(* Logix 5000 project; controller DispersionPlc vendor 1 type 14 code 108 rev 34.11; software revision 34.01; part 10 of 22 *)
(* tags used below, declared in another part *)
   ONS : BOOL[32];
   T4301Ons : BOOL[32];
   _JISdebug : DINT;
   _Placeholder : DINT;
   AFB : BOOL;
   AFI : BOOL;
   AirMakeup : TIMER;
   AirMakeup_BEAC : ALIAS FOR Local:1:O.Data[12].11;
   Cool_Setpoint_4301 : DINT;
   DispersionAlarms : BOOL[256];
   Emergency_Cool_4301 : BOOL;
   Emergency_Cool_4301_Reset : BOOL;
   Estop_Inx : ALIAS FOR Local:3:I.Data.3;
   Heat_Setpoint_4301 : DINT;
   HS_S51_2 : AStd_DiscreteInput;
   InxAlarms : BOOL[128];
   K2_Temperature_Alarm_Enable_Bit : BOOL;
   LS_T51_High : ALIAS FOR Local:1:I.Data[27].14;
   LVL_W2_High : ALIAS FOR Local:1:I.Data[1].22;
   LVL_W4_High : ALIAS FOR Local:1:I.Data[1].23;
   MaxHeatTmr4301 : TIMER;
   MIXER_A_4301_RUN : ALIAS FOR Local:1:O.Data[0].0;
   MMI_A_4301_01_RUN_PB : BOOL;
   MMI_A_4301_02_RUN_PB : BOOL;
   MMI_AIR_PURGE_4301_PB : BOOL;
   MMI_COOL_DISH_4301_PB : BOOL;
   MMI_COOL_VALVE_4301_PB : BOOL;
   MMI_Dispersion_Interlock_Bypass : BOOL;
   MMI_P_4301_RUN_PB : BOOL;
   MMI_T4301_AIR_PURGE_REQUEST : BOOL;
   MMI_T51_Level : INT;
   MMI_THINNING_LOADING_VALVE : BOOL;
   MMI_XV_4301_PB : BOOL;
   MMI_Z1H_4301_PB : BOOL;
   MMI_Z2H_4301_PB : BOOL;
   MMI_ZH3_4301_PB : BOOL;
   Ones4301 : DINT;
   OneShots2 : DINT;
   PID_T4301C : PID;
   PID_T4301H : PID;
   PS_AirMakeup : ALIAS FOR Local:1:I.Data[33].3;
   RG_T51 : REAL;
   RG_T51_AI_Holding : REAL;
   RG_T51_AI_Raw : INT;
   RG_T51_AI_Samples : DINT;
   RG_T51_Holding1 : REAL;
   RG_T51_Min_Tank_Value : INT;
   RG_T51_OffSet : REAL;
   RG_T51_REMAINDER : REAL;
   RG_T51_Sf : REAL;
   RM_High_Timer : TIMER;
   RM_Pump_P51_Aux : ALIAS FOR Local:1:I.Data[33].2;
   RM_Pump_P51_Run : ALIAS FOR Local:1:O.Data[13].0;
   RM_Pump_P51_Run_PB : ALIAS FOR Local:1:I.Data[40].0;
   RM_Pump_P51_Run_PB_2 : ALIAS FOR Local:1:I.Data[40].2;
   RM_Pump_P51_Stop_PB : ALIAS FOR Local:1:I.Data[40].1;
   RM_Pump_T51_Run_Lamp : ALIAS FOR Local:1:O.Data[12].2;
   RM_Pump_T51_Run_Lamp2 : ALIAS FOR Local:1:O.Data[0].20;
   RM_Tank_T51_Fill_Closed : ALIAS FOR Local:1:O.Data[12].10;
   RM_Tank_T51_Level_Lamp : ALIAS FOR Local:1:O.Data[12].5;
   RM_To_W2 : ALIAS FOR Local:1:I.Data[1].20;
   RM_To_W4 : ALIAS FOR Local:1:I.Data[1].21;
   SP : REAL;
   SPARE_I_1_4_6 : ALIAS FOR Local:1:I.Data[4].6;
   SPARE_O510 : ALIAS FOR Local:5:O.Data.10;
   SPARE_O600 : ALIAS FOR Local:6:O.Data.0;
   SPARE_O601 : ALIAS FOR Local:6:O.Data.1;
   SPARE_O602 : ALIAS FOR Local:6:O.Data.2;
   SPARE_O603 : ALIAS FOR Local:6:O.Data.3;
   SPARE_O604 : ALIAS FOR Local:6:O.Data.4;
   SPARE_O_13_1 : ALIAS FOR Local:13:O.Ch1Data;
   T4301_AIR_PURGE_REQUEST : BOOL;
   T4301_COOLING_OCCURED : BOOL;
   T4301_Cooling_On : BOOL;
   T4301_COOLING_OPERATION : BOOL;
   T4301_COOLING_TEMP : DINT;
   T4301_COOLING_VALVE_HMI : BOOL;
   T4301_DISCHARGE : BOOL;
   T4301_Heating_On : BOOL;
   T4301_HEATING_OPERATION : BOOL;
   T4301_HMI_Cooling : BOOL;
   T4301_HMI_Heating : BOOL;
   T4301_K : Kettle;
   T4301_Manual_AIR_PURGE_REQUEST : BOOL;
   T4301_Mixer : VFD;
   T4301_PID_Setpoints : PID[5];
   T4301_Pids_On : BOOL;
   T4301_PrePurgeTMR : TIMER;
   T4301_Purge_Complete : BOOL;
   T4301_Request_Cooling : BOOL;
   T4301_Request_Cooling_Tmr : TIMER[5];
   T4301_Request_Heating : BOOL;
   T4301_Request_Heating_Hold : BOOL;
   T4301_Request_Heating_Tmr : TIMER[5];
   T4301_Stop_Pids : BOOL;
   T4301ons2 : DINT;
   T4301Purge : Seq64;
   T51_Tank_Max_Lbs : REAL;
   TE_4301A : ALIAS FOR Local:8:I.Ch0Data;
   TempDifferenceCooling4301 : DINT;
   TempDifferenceCooling4301TMR : TIMER;
   testons : DINT;
   THINONS1 : BOOL;
   TOGGLE : BOOL;
   TRANS_PUMP_P_4301_RUN : ALIAS FOR Local:1:O.Data[0].1;
   W2_High_Level : BOOL;
   W4_High_Level : BOOL;
   XV_4301 : ALIAS FOR Local:5:O.Data.0;
   XV_S51_1 : AStd_VlvOC;
   XV_S51_4 : AStd_VlvOC;
(* MainProgram, continued *)

ROUTINE T4301   (* ladder *)
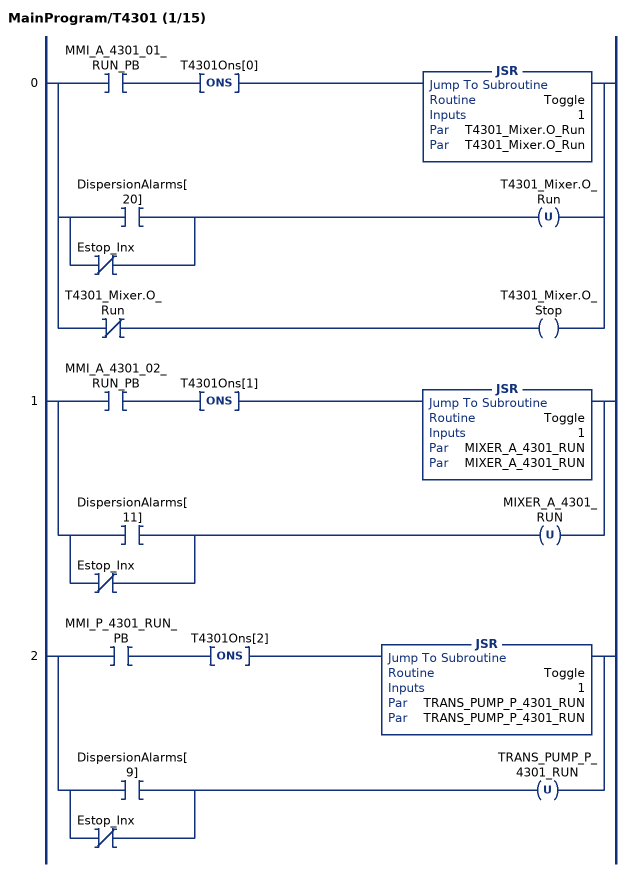
   0: [XIC(MMI_A_4301_01_RUN_PB) ONS(T4301Ons[0]) JSR(Toggle,1,T4301_Mixer.O_Run,T4301_Mixer.O_Run) ,[XIC(DispersionAlarms[20]) ,XIO(Estop_Inx) ] OTU(T4301_Mixer.O_Run) ,XIO(T4301_Mixer.O_Run) OTE(T4301_Mixer.O_Stop) ];
   1: [XIC(MMI_A_4301_02_RUN_PB) ONS(T4301Ons[1]) JSR(Toggle,1,MIXER_A_4301_RUN,MIXER_A_4301_RUN) ,[XIC(DispersionAlarms[11]) ,XIO(Estop_Inx) ] OTU(MIXER_A_4301_RUN) ];
   2: [XIC(MMI_P_4301_RUN_PB) ONS(T4301Ons[2]) JSR(Toggle,1,TRANS_PUMP_P_4301_RUN,TRANS_PUMP_P_4301_RUN) ,[XIC(DispersionAlarms[9]) ,XIO(Estop_Inx) ] OTU(TRANS_PUMP_P_4301_RUN) ];
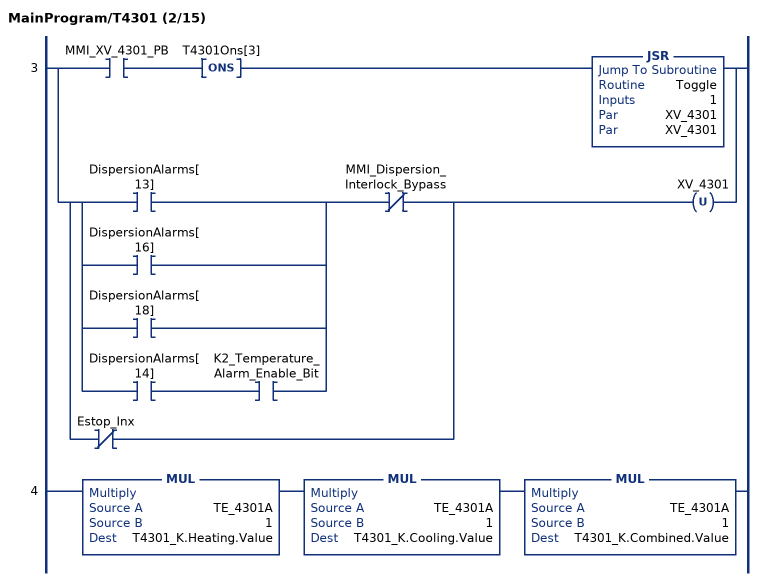
   3: [XIC(MMI_XV_4301_PB) ONS(T4301Ons[3]) JSR(Toggle,1,XV_4301,XV_4301) ,[[XIC(DispersionAlarms[13]) ,XIC(DispersionAlarms[16]) ,XIC(DispersionAlarms[18]) ,XIC(DispersionAlarms[14]) XIC(K2_Temperature_Alarm_Enable_Bit) ] XIO(MMI_Dispersion_Interlock_Bypass) ,XIO(Estop_Inx) ] OTU(XV_4301) ];
   4: MUL(TE_4301A,1,T4301_K.Heating.Value)MUL(TE_4301A,1,T4301_K.Cooling.Value)MUL(TE_4301A,1,T4301_K.Combined.Value);
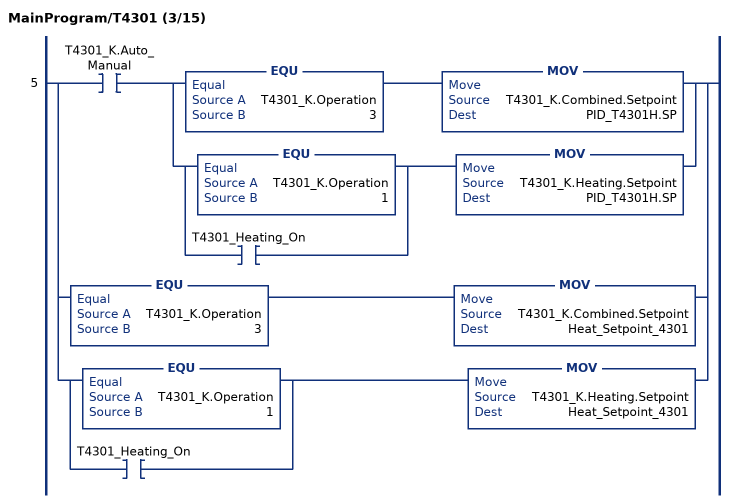
   5: [XIC(T4301_K.Auto_Manual) [EQU(T4301_K.Operation,3) MOV(T4301_K.Combined.Setpoint,PID_T4301H.SP) ,[EQU(T4301_K.Operation,1) ,XIC(T4301_Heating_On) ] MOV(T4301_K.Heating.Setpoint,PID_T4301H.SP) ] ,[EQU(T4301_K.Operation,3) MOV(T4301_K.Combined.Setpoint,Heat_Setpoint_4301) ,[EQU(T4301_K.Operation,1) ,XIC(T4301_Heating_On) ] MOV(T4301_K.Heating.Setpoint,Heat_Setpoint_4301) ] ];
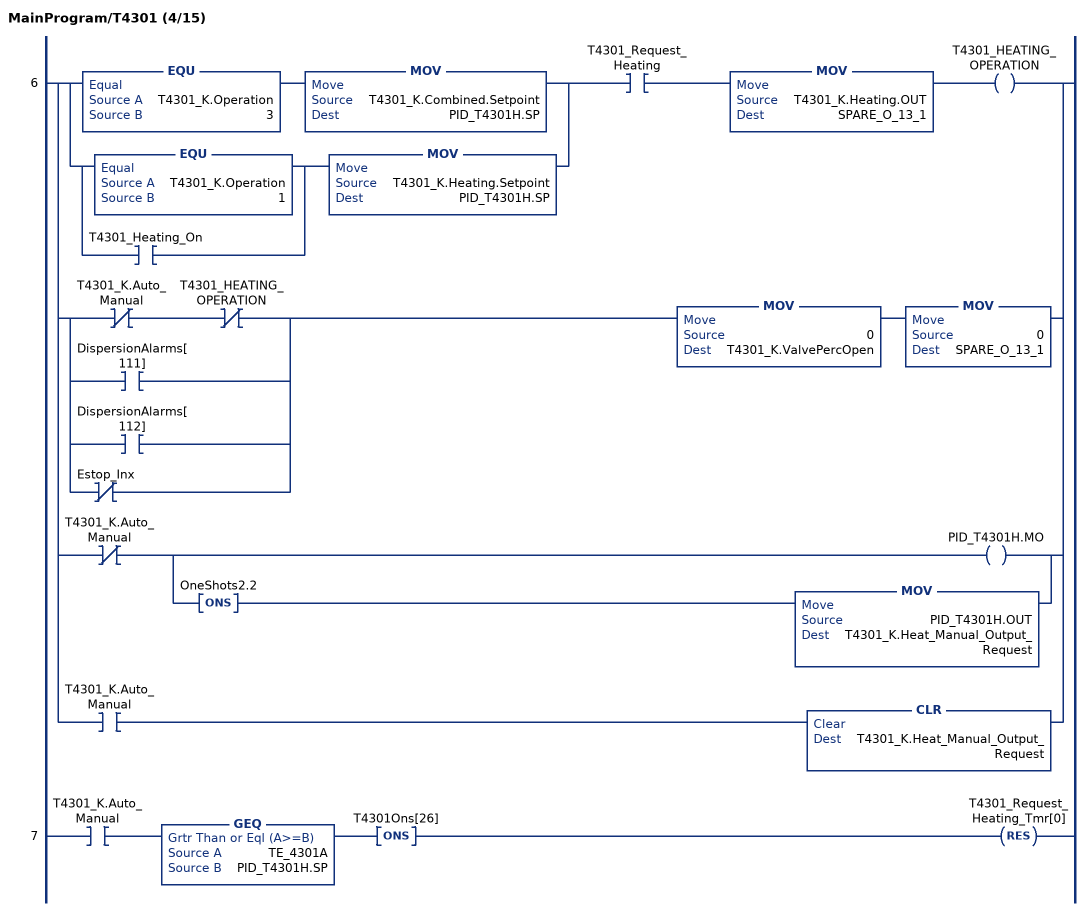
   6: [[EQU(T4301_K.Operation,3) MOV(T4301_K.Combined.Setpoint,PID_T4301H.SP) ,[EQU(T4301_K.Operation,1) ,XIC(T4301_Heating_On) ] MOV(T4301_K.Heating.Setpoint,PID_T4301H.SP) ] XIC(T4301_Request_Heating) MOV(T4301_K.Heating.OUT,SPARE_O_13_1) OTE(T4301_HEATING_OPERATION) ,[XIO(T4301_K.Auto_Manual) XIO(T4301_HEATING_OPERATION) ,[XIC(DispersionAlarms[111]) ,XIC(DispersionAlarms[112]) ,XIO(Estop_Inx) ] ] MOV(0,T4301_K.ValvePercOpen) MOV(0,SPARE_O_13_1) ,[XIO(T4301_K.Auto_Manual) [OTE(PID_T4301H.MO) ,ONS(OneShots2.2) MOV(PID_T4301H.OUT,T4301_K.Heat_Manual_Output_Request) ] ,XIC(T4301_K.Auto_Manual) CLR(T4301_K.Heat_Manual_Output_Request) ] ];
   7: XIC(T4301_K.Auto_Manual)GEQ(TE_4301A,PID_T4301H.SP)ONS(T4301Ons[26])RES(T4301_Request_Heating_Tmr[0]);
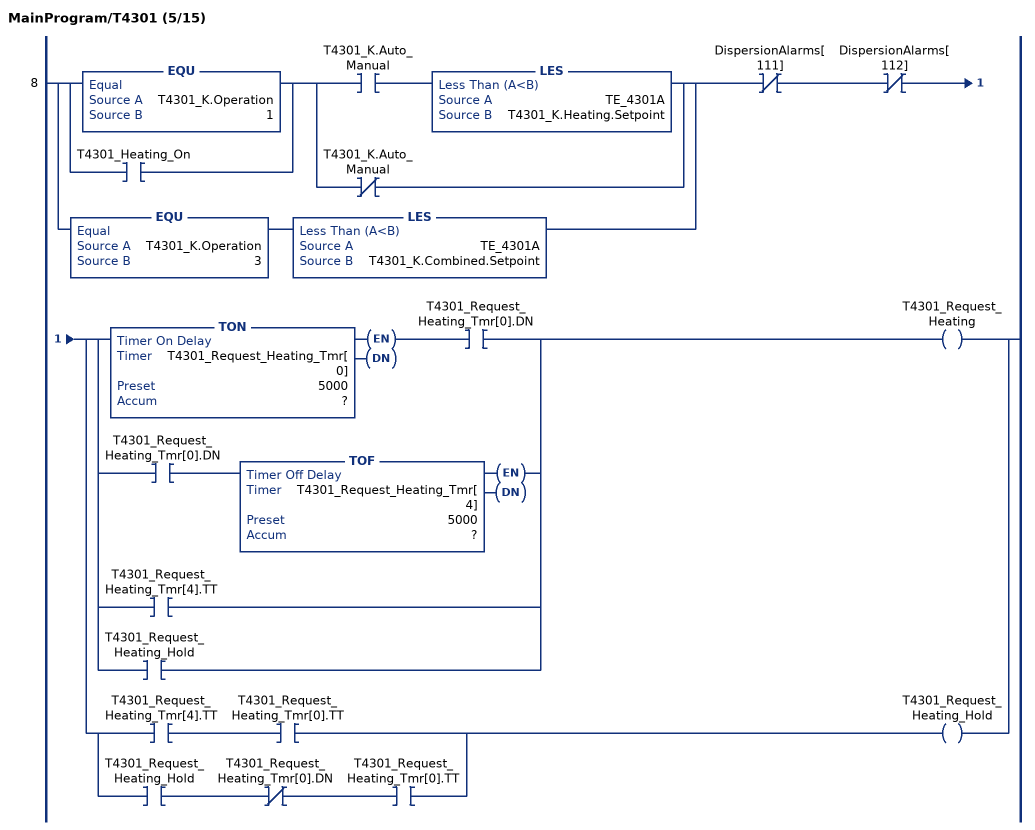
   8: [[EQU(T4301_K.Operation,1) ,XIC(T4301_Heating_On) ] [XIC(T4301_K.Auto_Manual) LES(TE_4301A,T4301_K.Heating.Setpoint) ,XIO(T4301_K.Auto_Manual) ] ,EQU(T4301_K.Operation,3) LES(TE_4301A,T4301_K.Combined.Setpoint) ]XIO(DispersionAlarms[111])XIO(DispersionAlarms[112])[[TON(T4301_Request_Heating_Tmr[0],?,?) XIC(T4301_Request_Heating_Tmr[0].DN) ,XIC(T4301_Request_Heating_Tmr[0].DN) TOF(T4301_Request_Heating_Tmr[4],?,?) ,XIC(T4301_Request_Heating_Tmr[4].TT) ,XIC(T4301_Request_Heating_Hold) ] OTE(T4301_Request_Heating) ,[XIC(T4301_Request_Heating_Tmr[4].TT) XIC(T4301_Request_Heating_Tmr[0].TT) ,XIC(T4301_Request_Heating_Hold) XIO(T4301_Request_Heating_Tmr[0].DN) XIC(T4301_Request_Heating_Tmr[0].TT) ] OTE(T4301_Request_Heating_Hold) ];
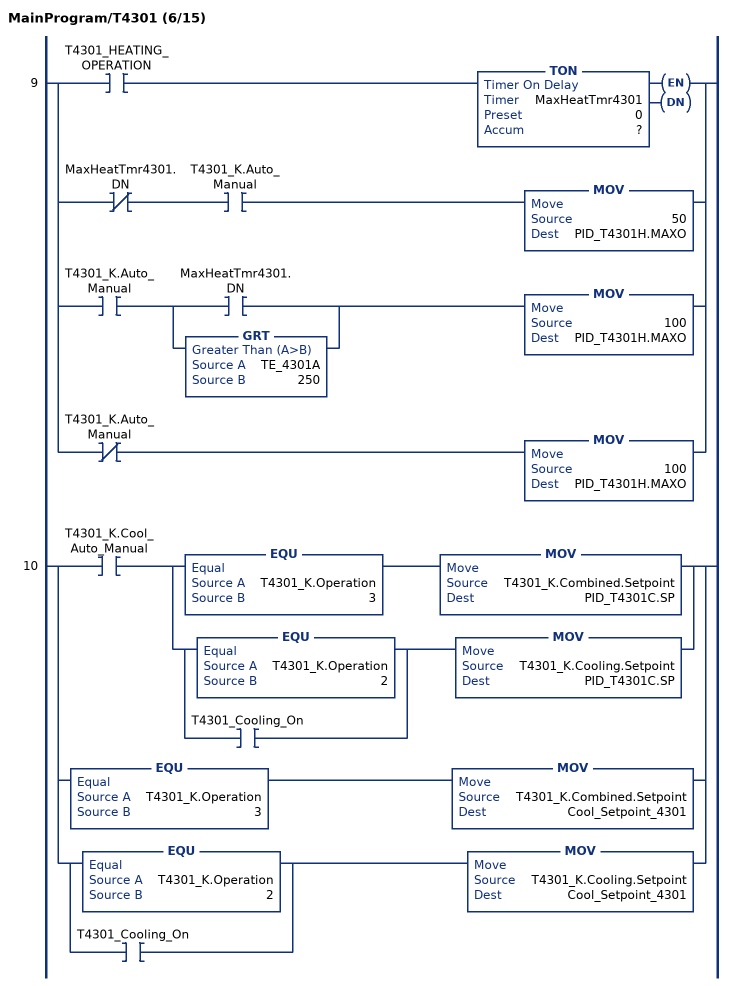
   9: [XIC(T4301_HEATING_OPERATION) TON(MaxHeatTmr4301,?,?) ,XIO(MaxHeatTmr4301.DN) XIC(T4301_K.Auto_Manual) MOV(50,PID_T4301H.MAXO) ,XIC(T4301_K.Auto_Manual) [XIC(MaxHeatTmr4301.DN) ,GRT(TE_4301A,250) ] MOV(100,PID_T4301H.MAXO) ,XIO(T4301_K.Auto_Manual) MOV(100,PID_T4301H.MAXO) ];
   10: [XIC(T4301_K.Cool_Auto_Manual) [EQU(T4301_K.Operation,3) MOV(T4301_K.Combined.Setpoint,PID_T4301C.SP) ,[EQU(T4301_K.Operation,2) ,XIC(T4301_Cooling_On) ] MOV(T4301_K.Cooling.Setpoint,PID_T4301C.SP) ] ,[EQU(T4301_K.Operation,3) MOV(T4301_K.Combined.Setpoint,Cool_Setpoint_4301) ,[EQU(T4301_K.Operation,2) ,XIC(T4301_Cooling_On) ] MOV(T4301_K.Cooling.Setpoint,Cool_Setpoint_4301) ] ];
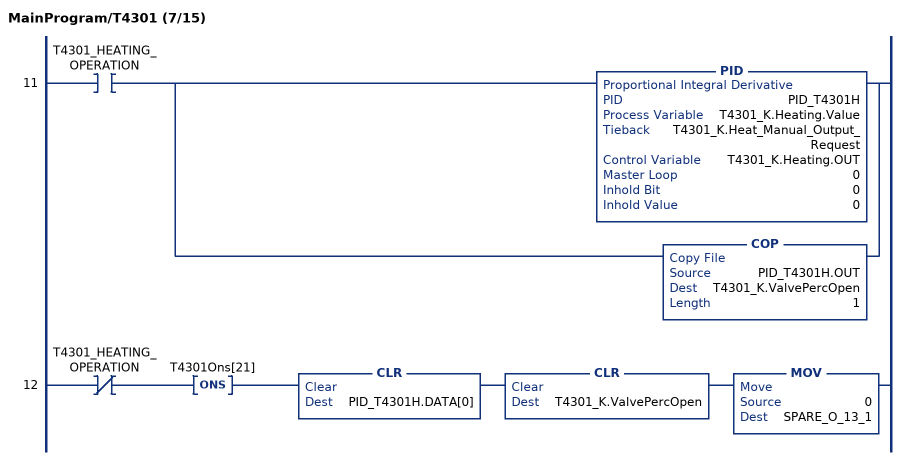
   11: XIC(T4301_HEATING_OPERATION)[PID(PID_T4301H,T4301_K.Heating.Value,T4301_K.Heat_Manual_Output_Request,T4301_K.Heating.OUT,0,0,0) ,COP(PID_T4301H.OUT,T4301_K.ValvePercOpen,1) ];
   12: XIO(T4301_HEATING_OPERATION)ONS(T4301Ons[21])CLR(PID_T4301H.DATA[0])CLR(T4301_K.ValvePercOpen)MOV(0,SPARE_O_13_1);
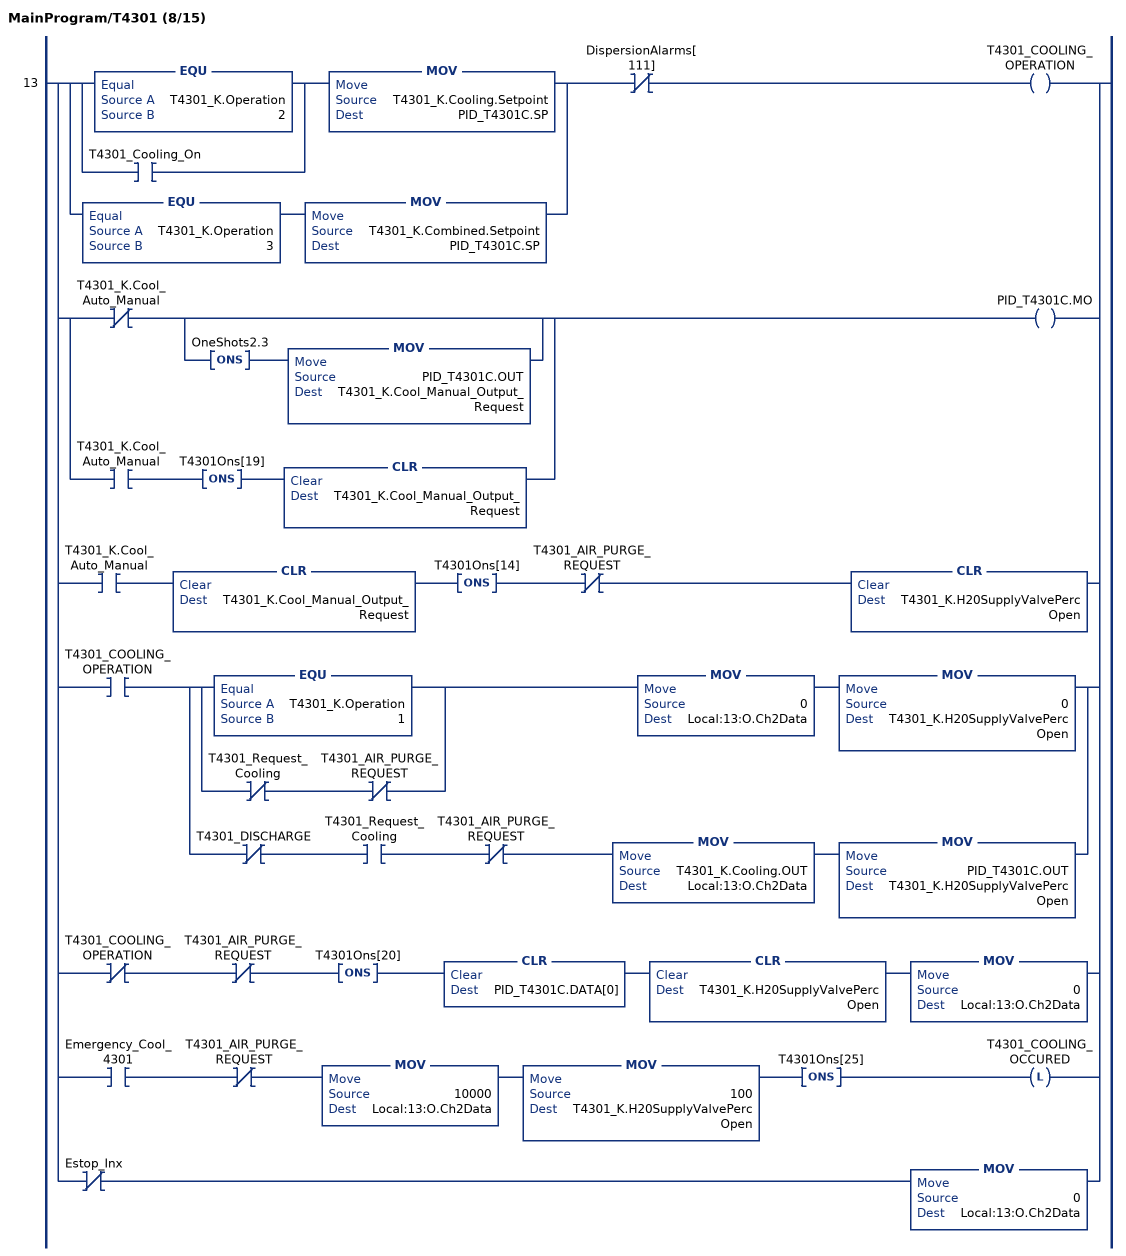
   13: [[[EQU(T4301_K.Operation,2) ,XIC(T4301_Cooling_On) ] MOV(T4301_K.Cooling.Setpoint,PID_T4301C.SP) ,EQU(T4301_K.Operation,3) MOV(T4301_K.Combined.Setpoint,PID_T4301C.SP) ] XIO(DispersionAlarms[111]) OTE(T4301_COOLING_OPERATION) ,[[XIO(T4301_K.Cool_Auto_Manual) [,ONS(OneShots2.3) MOV(PID_T4301C.OUT,T4301_K.Cool_Manual_Output_Request) ] ,XIC(T4301_K.Cool_Auto_Manual) ONS(T4301Ons[19]) CLR(T4301_K.Cool_Manual_Output_Request) ] OTE(PID_T4301C.MO) ,XIC(T4301_K.Cool_Auto_Manual) CLR(T4301_K.Cool_Manual_Output_Request) ONS(T4301Ons[14]) XIO(T4301_AIR_PURGE_REQUEST) CLR(T4301_K.H20SupplyValvePercOpen) ] ,XIC(T4301_COOLING_OPERATION) [[EQU(T4301_K.Operation,1) ,XIO(T4301_Request_Cooling) XIO(T4301_AIR_PURGE_REQUEST) ] MOV(0,Local:13:O.Ch2Data) MOV(0,T4301_K.H20SupplyValvePercOpen) ,XIO(T4301_DISCHARGE) XIC(T4301_Request_Cooling) XIO(T4301_AIR_PURGE_REQUEST) MOV(T4301_K.Cooling.OUT,Local:13:O.Ch2Data) MOV(PID_T4301C.OUT,T4301_K.H20SupplyValvePercOpen) ] ,XIO(T4301_COOLING_OPERATION) XIO(T4301_AIR_PURGE_REQUEST) ONS(T4301Ons[20]) CLR(PID_T4301C.DATA[0]) CLR(T4301_K.H20SupplyValvePercOpen) MOV(0,Local:13:O.Ch2Data) ,XIC(Emergency_Cool_4301) XIO(T4301_AIR_PURGE_REQUEST) MOV(10000,Local:13:O.Ch2Data) MOV(100,T4301_K.H20SupplyValvePercOpen) ONS(T4301Ons[25]) OTL(T4301_COOLING_OCCURED) ,XIO(Estop_Inx) MOV(0,Local:13:O.Ch2Data) ];
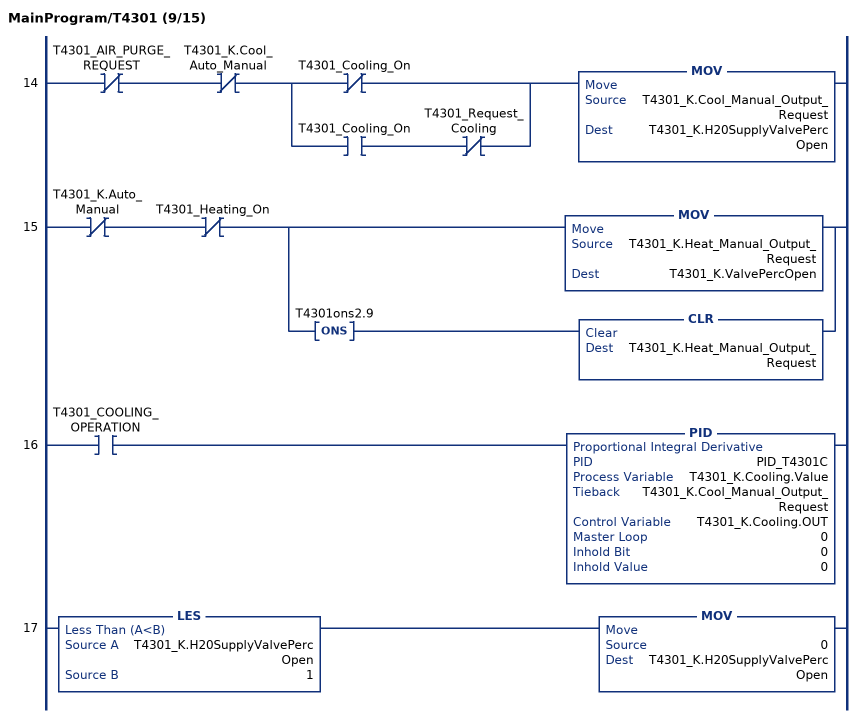
   14: XIO(T4301_AIR_PURGE_REQUEST)XIO(T4301_K.Cool_Auto_Manual)[XIO(T4301_Cooling_On) ,XIC(T4301_Cooling_On) XIO(T4301_Request_Cooling) ]MOV(T4301_K.Cool_Manual_Output_Request,T4301_K.H20SupplyValvePercOpen);
   15: XIO(T4301_K.Auto_Manual)XIO(T4301_Heating_On)[MOV(T4301_K.Heat_Manual_Output_Request,T4301_K.ValvePercOpen) ,ONS(T4301ons2.9) CLR(T4301_K.Heat_Manual_Output_Request) ];
   16: XIC(T4301_COOLING_OPERATION)PID(PID_T4301C,T4301_K.Cooling.Value,T4301_K.Cool_Manual_Output_Request,T4301_K.Cooling.OUT,0,0,0);
   17: LES(T4301_K.H20SupplyValvePercOpen,1)MOV(0,T4301_K.H20SupplyValvePercOpen);
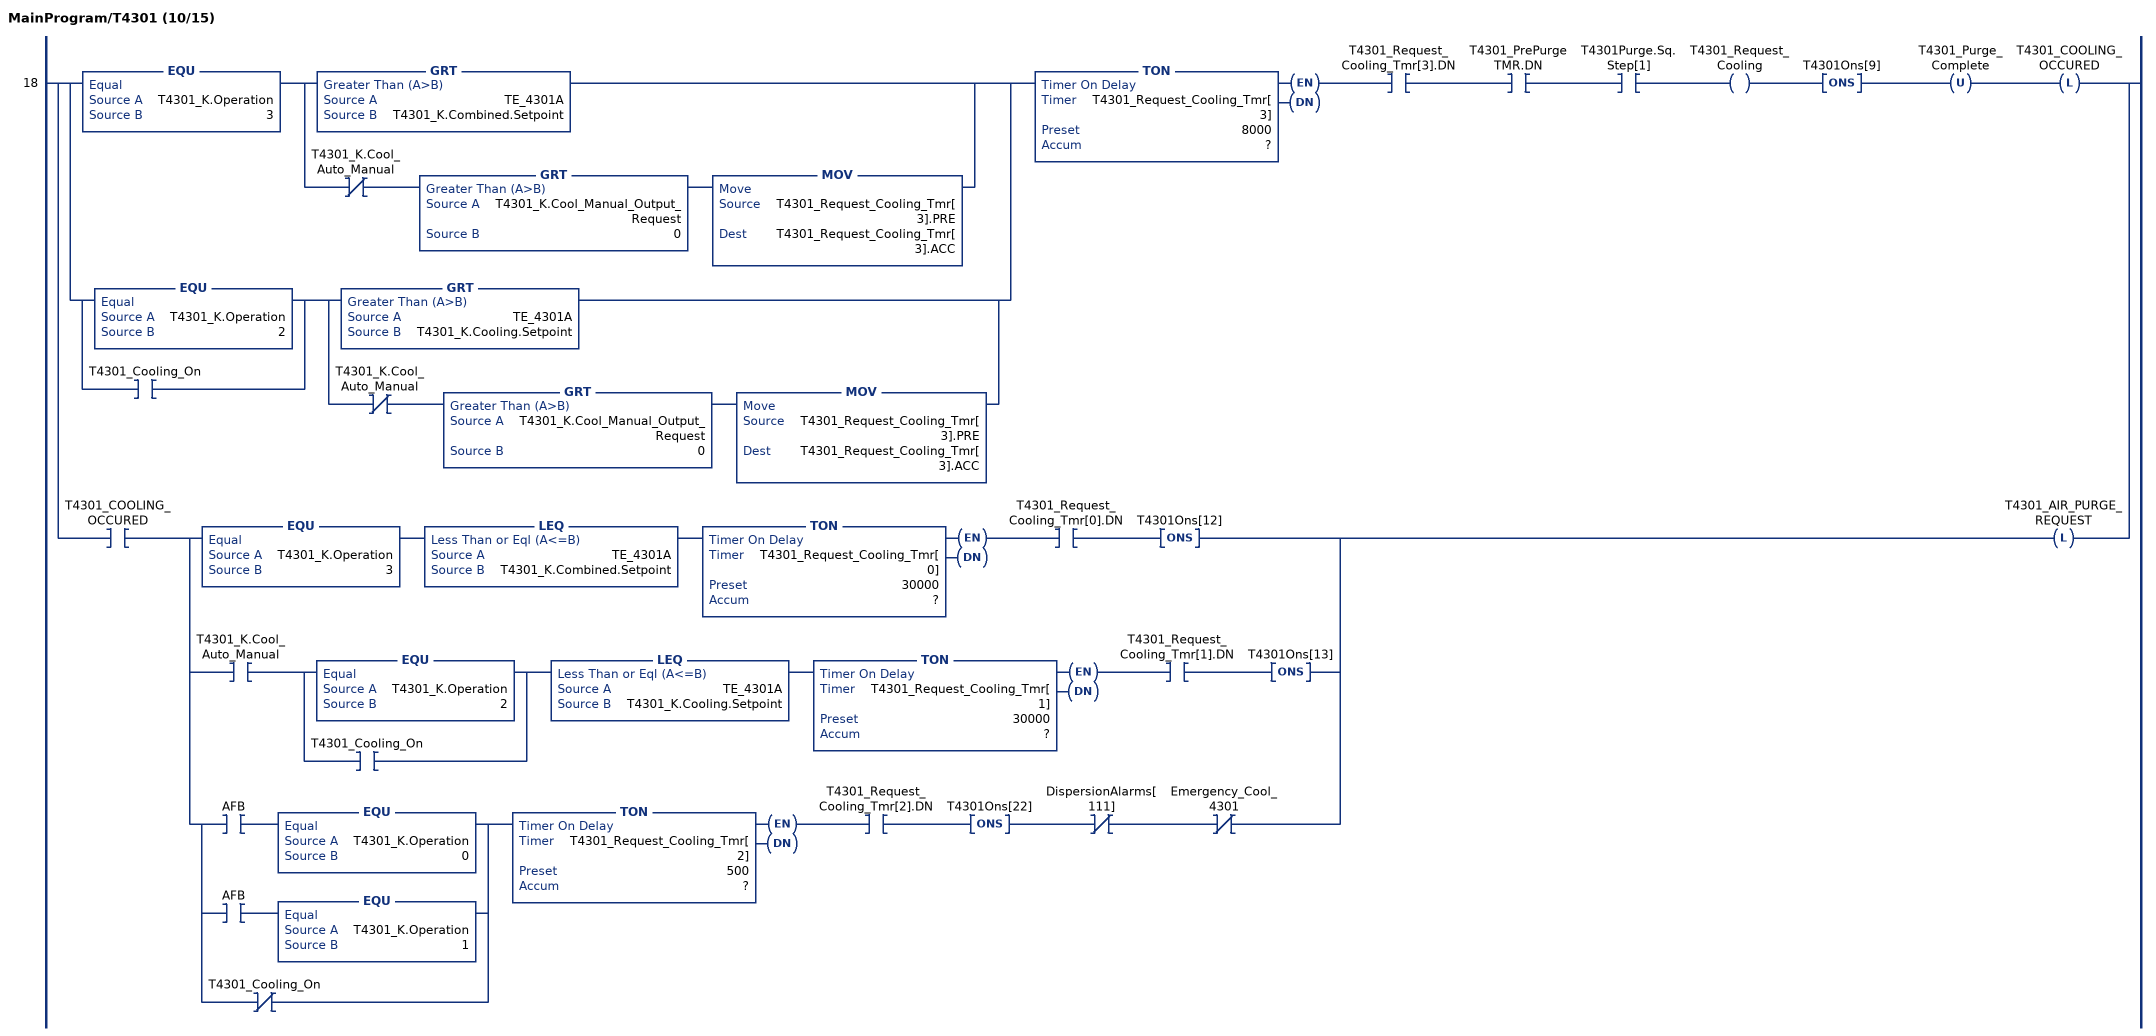
   18: [[EQU(T4301_K.Operation,3) [GRT(TE_4301A,T4301_K.Combined.Setpoint) ,XIO(T4301_K.Cool_Auto_Manual) GRT(T4301_K.Cool_Manual_Output_Request,0) MOV(T4301_Request_Cooling_Tmr[3].PRE,T4301_Request_Cooling_Tmr[3].ACC) ] ,[EQU(T4301_K.Operation,2) ,XIC(T4301_Cooling_On) ] [GRT(TE_4301A,T4301_K.Cooling.Setpoint) ,XIO(T4301_K.Cool_Auto_Manual) GRT(T4301_K.Cool_Manual_Output_Request,0) MOV(T4301_Request_Cooling_Tmr[3].PRE,T4301_Request_Cooling_Tmr[3].ACC) ] ] TON(T4301_Request_Cooling_Tmr[3],?,?) XIC(T4301_Request_Cooling_Tmr[3].DN) XIC(T4301_PrePurgeTMR.DN) XIC(T4301Purge.Sq.Step[1]) OTE(T4301_Request_Cooling) ONS(T4301Ons[9]) OTU(T4301_Purge_Complete) OTL(T4301_COOLING_OCCURED) ,XIC(T4301_COOLING_OCCURED) [EQU(T4301_K.Operation,3) LEQ(TE_4301A,T4301_K.Combined.Setpoint) TON(T4301_Request_Cooling_Tmr[0],?,?) XIC(T4301_Request_Cooling_Tmr[0].DN) ONS(T4301Ons[12]) ,XIC(T4301_K.Cool_Auto_Manual) [EQU(T4301_K.Operation,2) ,XIC(T4301_Cooling_On) ] LEQ(TE_4301A,T4301_K.Cooling.Setpoint) TON(T4301_Request_Cooling_Tmr[1],?,?) XIC(T4301_Request_Cooling_Tmr[1].DN) ONS(T4301Ons[13]) ,[XIC(AFB) EQU(T4301_K.Operation,0) ,XIC(AFB) EQU(T4301_K.Operation,1) ,XIO(T4301_Cooling_On) ] TON(T4301_Request_Cooling_Tmr[2],?,?) XIC(T4301_Request_Cooling_Tmr[2].DN) ONS(T4301Ons[22]) XIO(DispersionAlarms[111]) XIO(Emergency_Cool_4301) ] OTL(T4301_AIR_PURGE_REQUEST) ];
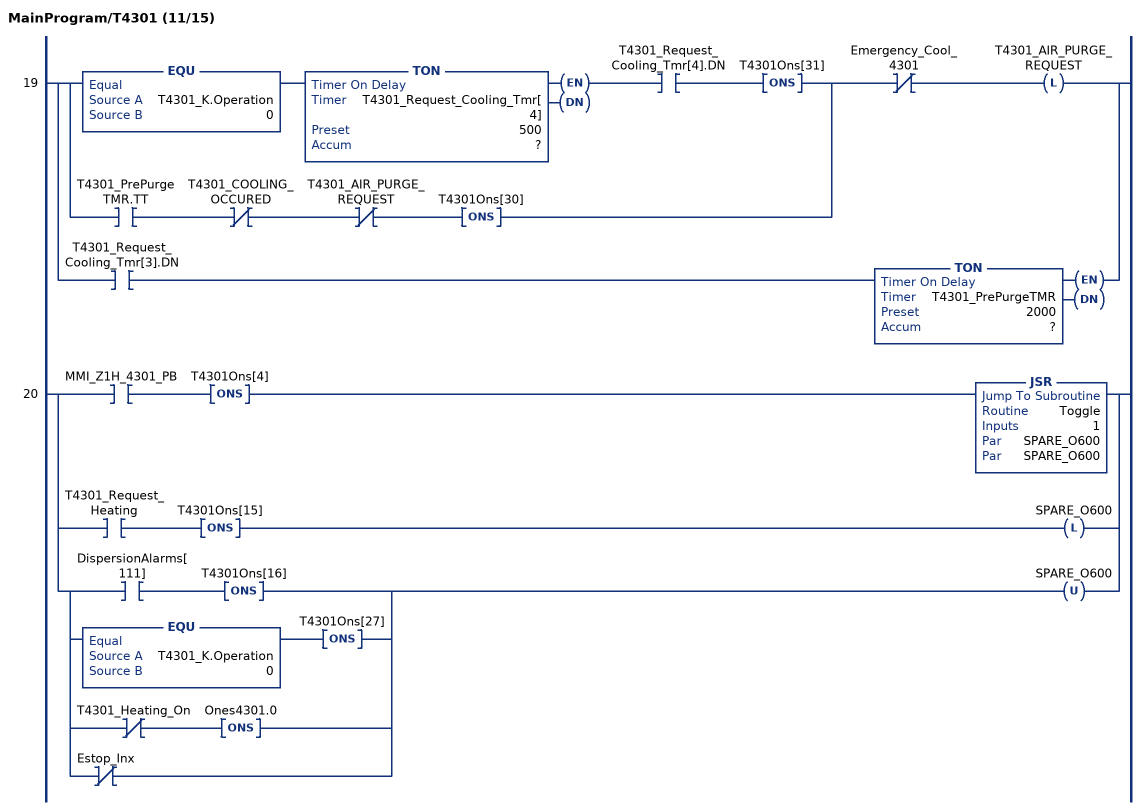
   19: [[EQU(T4301_K.Operation,0) TON(T4301_Request_Cooling_Tmr[4],?,?) XIC(T4301_Request_Cooling_Tmr[4].DN) ONS(T4301Ons[31]) ,XIC(T4301_PrePurgeTMR.TT) XIO(T4301_COOLING_OCCURED) XIO(T4301_AIR_PURGE_REQUEST) ONS(T4301Ons[30]) ] XIO(Emergency_Cool_4301) OTL(T4301_AIR_PURGE_REQUEST) ,XIC(T4301_Request_Cooling_Tmr[3].DN) TON(T4301_PrePurgeTMR,?,?) ];
   20: [XIC(MMI_Z1H_4301_PB) ONS(T4301Ons[4]) JSR(Toggle,1,SPARE_O600,SPARE_O600) ,XIC(T4301_Request_Heating) ONS(T4301Ons[15]) OTL(SPARE_O600) ,[XIC(DispersionAlarms[111]) ONS(T4301Ons[16]) ,[EQU(T4301_K.Operation,0) ONS(T4301Ons[27]) ,XIO(T4301_Heating_On) ONS(Ones4301.0) ] ,XIO(Estop_Inx) ] OTU(SPARE_O600) ];
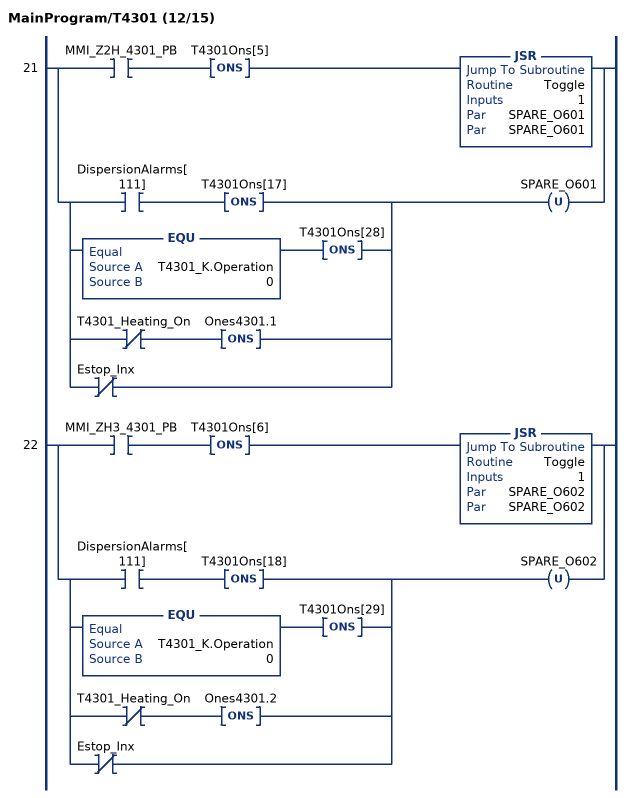
   21: [XIC(MMI_Z2H_4301_PB) ONS(T4301Ons[5]) JSR(Toggle,1,SPARE_O601,SPARE_O601) ,[XIC(DispersionAlarms[111]) ONS(T4301Ons[17]) ,[EQU(T4301_K.Operation,0) ONS(T4301Ons[28]) ,XIO(T4301_Heating_On) ONS(Ones4301.1) ] ,XIO(Estop_Inx) ] OTU(SPARE_O601) ];
   22: [XIC(MMI_ZH3_4301_PB) ONS(T4301Ons[6]) JSR(Toggle,1,SPARE_O602,SPARE_O602) ,[XIC(DispersionAlarms[111]) ONS(T4301Ons[18]) ,[EQU(T4301_K.Operation,0) ONS(T4301Ons[29]) ,XIO(T4301_Heating_On) ONS(Ones4301.2) ] ,XIO(Estop_Inx) ] OTU(SPARE_O602) ];
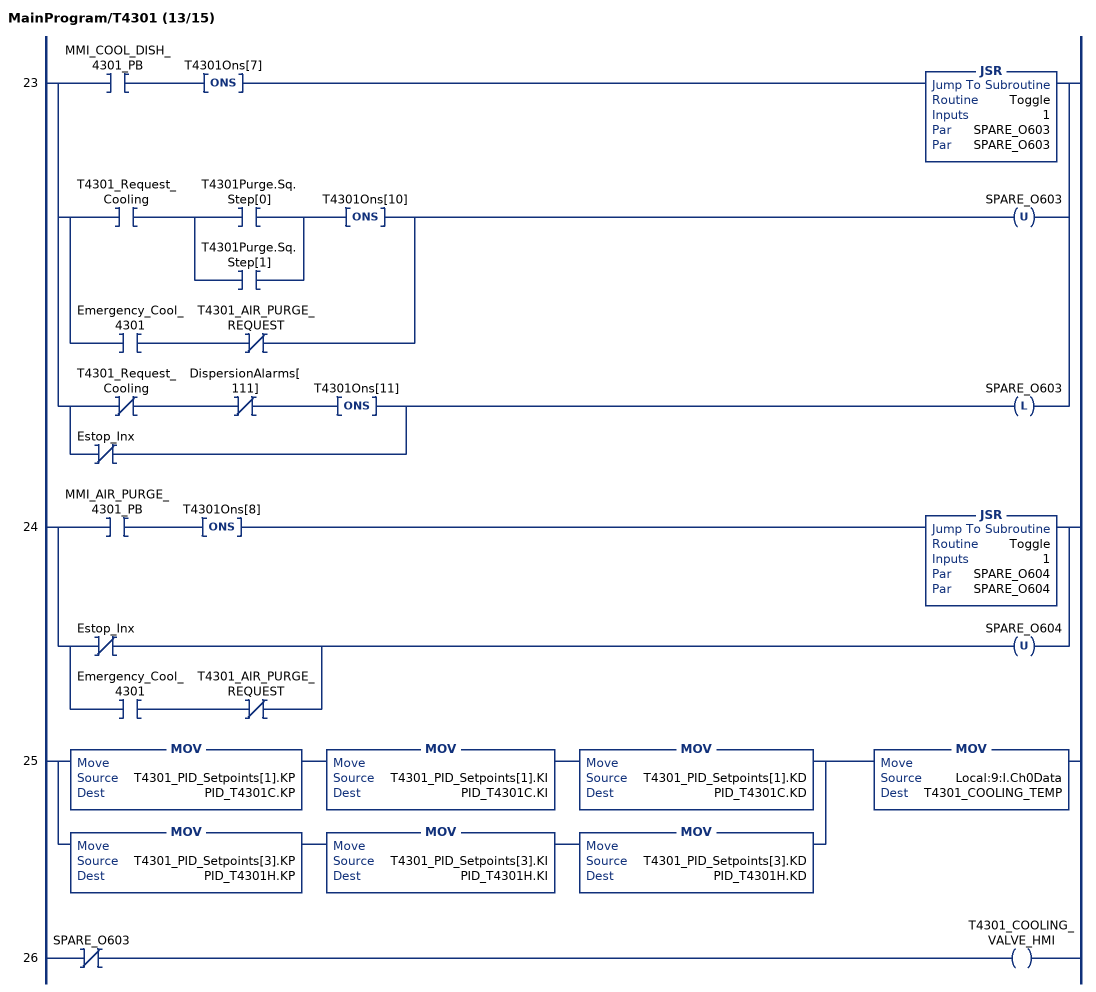
   23: [XIC(MMI_COOL_DISH_4301_PB) ONS(T4301Ons[7]) JSR(Toggle,1,SPARE_O603,SPARE_O603) ,[XIC(T4301_Request_Cooling) [XIC(T4301Purge.Sq.Step[0]) ,XIC(T4301Purge.Sq.Step[1]) ] ONS(T4301Ons[10]) ,XIC(Emergency_Cool_4301) XIO(T4301_AIR_PURGE_REQUEST) ] OTU(SPARE_O603) ,[XIO(T4301_Request_Cooling) XIO(DispersionAlarms[111]) ONS(T4301Ons[11]) ,XIO(Estop_Inx) ] OTL(SPARE_O603) ];
   24: [XIC(MMI_AIR_PURGE_4301_PB) ONS(T4301Ons[8]) JSR(Toggle,1,SPARE_O604,SPARE_O604) ,[XIO(Estop_Inx) ,XIC(Emergency_Cool_4301) XIO(T4301_AIR_PURGE_REQUEST) ] OTU(SPARE_O604) ];
   25: [MOV(T4301_PID_Setpoints[1].KP,PID_T4301C.KP) MOV(T4301_PID_Setpoints[1].KI,PID_T4301C.KI) MOV(T4301_PID_Setpoints[1].KD,PID_T4301C.KD) ,MOV(T4301_PID_Setpoints[3].KP,PID_T4301H.KP) MOV(T4301_PID_Setpoints[3].KI,PID_T4301H.KI) MOV(T4301_PID_Setpoints[3].KD,PID_T4301H.KD) ]MOV(Local:9:I.Ch0Data,T4301_COOLING_TEMP);
   26: XIO(SPARE_O603)OTE(T4301_COOLING_VALVE_HMI);
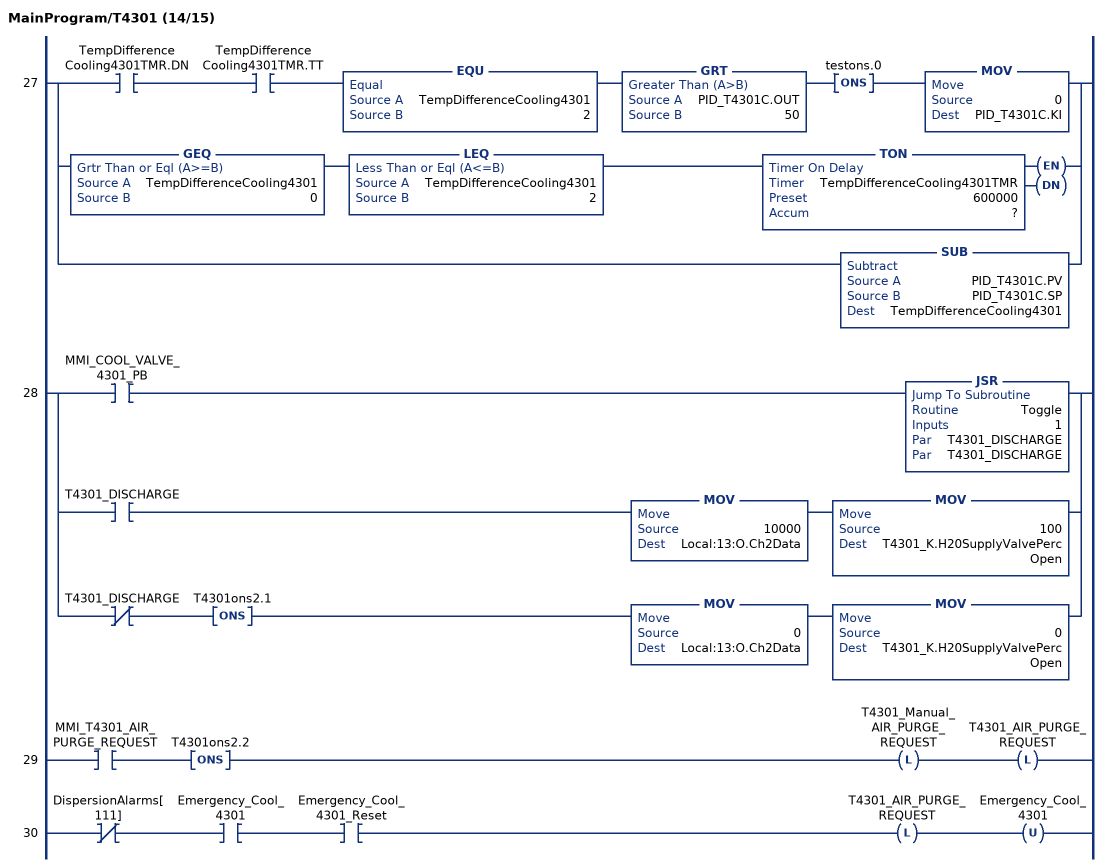
   27: [XIC(TempDifferenceCooling4301TMR.DN) XIC(TempDifferenceCooling4301TMR.TT) EQU(TempDifferenceCooling4301,2) GRT(PID_T4301C.OUT,50) ONS(testons.0) MOV(0,PID_T4301C.KI) ,GEQ(TempDifferenceCooling4301,0) LEQ(TempDifferenceCooling4301,2) TON(TempDifferenceCooling4301TMR,?,?) ,SUB(PID_T4301C.PV,PID_T4301C.SP,TempDifferenceCooling4301) ];
   28: [XIC(MMI_COOL_VALVE_4301_PB) JSR(Toggle,1,T4301_DISCHARGE,T4301_DISCHARGE) ,XIC(T4301_DISCHARGE) MOV(10000,Local:13:O.Ch2Data) MOV(100,T4301_K.H20SupplyValvePercOpen) ,XIO(T4301_DISCHARGE) ONS(T4301ons2.1) MOV(0,Local:13:O.Ch2Data) MOV(0,T4301_K.H20SupplyValvePercOpen) ];
   29: XIC(MMI_T4301_AIR_PURGE_REQUEST)ONS(T4301ons2.2)OTL(T4301_Manual_AIR_PURGE_REQUEST)OTL(T4301_AIR_PURGE_REQUEST);
   30: XIO(DispersionAlarms[111])XIC(Emergency_Cool_4301)XIC(Emergency_Cool_4301_Reset)OTL(T4301_AIR_PURGE_REQUEST)OTU(Emergency_Cool_4301);
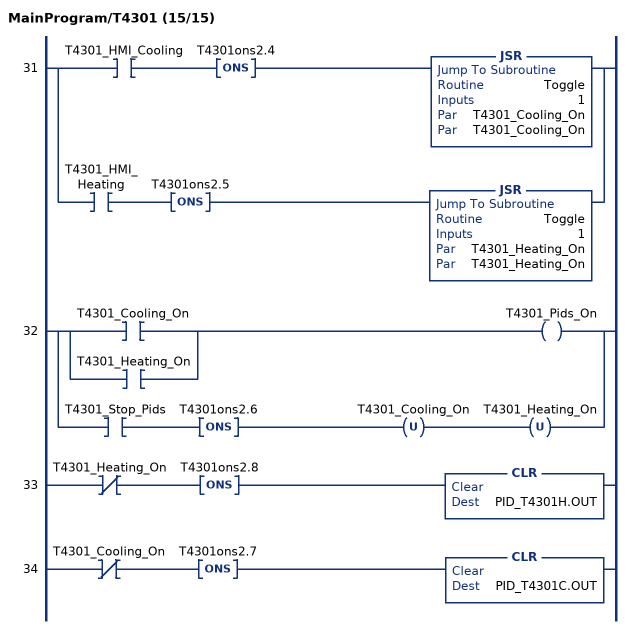
   31: [XIC(T4301_HMI_Cooling) ONS(T4301ons2.4) JSR(Toggle,1,T4301_Cooling_On,T4301_Cooling_On) ,XIC(T4301_HMI_Heating) ONS(T4301ons2.5) JSR(Toggle,1,T4301_Heating_On,T4301_Heating_On) ];
   32: [[XIC(T4301_Cooling_On) ,XIC(T4301_Heating_On) ] OTE(T4301_Pids_On) ,XIC(T4301_Stop_Pids) ONS(T4301ons2.6) OTU(T4301_Cooling_On) OTU(T4301_Heating_On) ];
   33: XIO(T4301_Heating_On)ONS(T4301ons2.8)CLR(PID_T4301H.OUT);
   34: XIO(T4301_Cooling_On)ONS(T4301ons2.7)CLR(PID_T4301C.OUT);
END_ROUTINE

ROUTINE T51   (* ladder *)
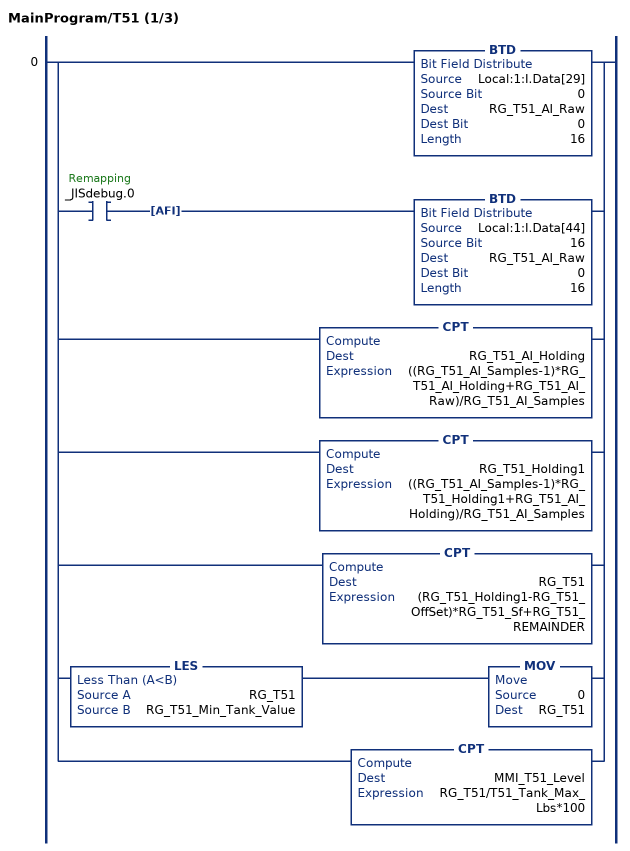
   0: [BTD(Local:1:I.Data[29],0,RG_T51_AI_Raw,0,16) ,XIC(_JISdebug.0) AFI() BTD(Local:1:I.Data[44],16,RG_T51_AI_Raw,0,16) ,CPT(RG_T51_AI_Holding,((RG_T51_AI_Samples-1)*RG_T51_AI_Holding+RG_T51_AI_Raw)/RG_T51_AI_Samples) ,CPT(RG_T51_Holding1,((RG_T51_AI_Samples-1)*RG_T51_Holding1+RG_T51_AI_Holding)/RG_T51_AI_Samples) ,CPT(RG_T51,(RG_T51_Holding1-RG_T51_OffSet)*RG_T51_Sf+RG_T51_REMAINDER) ,LES(RG_T51,RG_T51_Min_Tank_Value) MOV(0,RG_T51) ,CPT(MMI_T51_Level,RG_T51/T51_Tank_Max_Lbs*100) ];
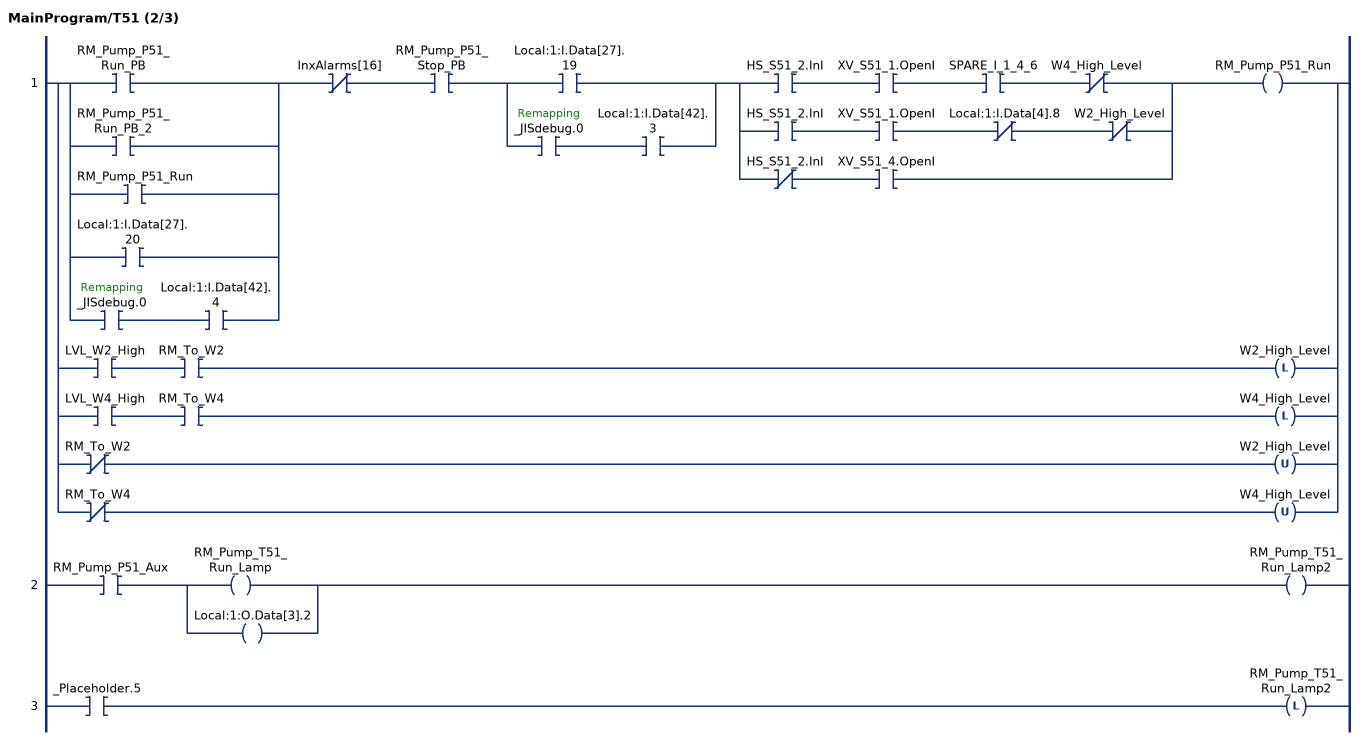
   1: [[XIC(RM_Pump_P51_Run_PB) ,XIC(RM_Pump_P51_Run_PB_2) ,XIC(RM_Pump_P51_Run) ,XIC(Local:1:I.Data[27].20) ,XIC(_JISdebug.0) XIC(Local:1:I.Data[42].4) ] XIO(InxAlarms[16]) XIC(RM_Pump_P51_Stop_PB) [XIC(Local:1:I.Data[27].19) ,XIC(_JISdebug.0) XIC(Local:1:I.Data[42].3) ] [XIC(HS_S51_2.InI) XIC(XV_S51_1.OpenI) XIC(SPARE_I_1_4_6) XIO(W4_High_Level) ,XIC(HS_S51_2.InI) XIC(XV_S51_1.OpenI) XIO(Local:1:I.Data[4].8) XIO(W2_High_Level) ,XIO(HS_S51_2.InI) XIC(XV_S51_4.OpenI) ] OTE(RM_Pump_P51_Run) ,[XIC(LVL_W2_High) XIC(RM_To_W2) OTL(W2_High_Level) ,XIC(LVL_W4_High) XIC(RM_To_W4) OTL(W4_High_Level) ] ,[XIO(RM_To_W2) OTU(W2_High_Level) ,XIO(RM_To_W4) OTU(W4_High_Level) ] ];
   2: XIC(RM_Pump_P51_Aux)[OTE(RM_Pump_T51_Run_Lamp) ,OTE(Local:1:O.Data[3].2) ]OTE(RM_Pump_T51_Run_Lamp2);
   3: XIC(_Placeholder.5)OTL(RM_Pump_T51_Run_Lamp2);
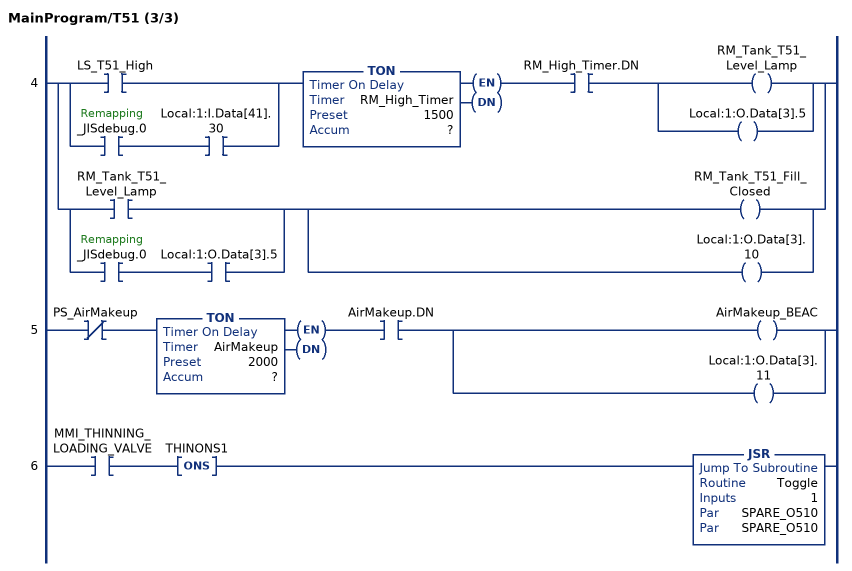
   4: [[XIC(LS_T51_High) ,XIC(_JISdebug.0) XIC(Local:1:I.Data[41].30) ] TON(RM_High_Timer,?,?) XIC(RM_High_Timer.DN) [OTE(RM_Tank_T51_Level_Lamp) ,OTE(Local:1:O.Data[3].5) ] ,[XIC(RM_Tank_T51_Level_Lamp) ,XIC(_JISdebug.0) XIC(Local:1:O.Data[3].5) ] [OTE(RM_Tank_T51_Fill_Closed) ,OTE(Local:1:O.Data[3].10) ] ];
   5: XIO(PS_AirMakeup)TON(AirMakeup,?,?)XIC(AirMakeup.DN)[OTE(AirMakeup_BEAC) ,OTE(Local:1:O.Data[3].11) ];
   6: XIC(MMI_THINNING_LOADING_VALVE)ONS(THINONS1)JSR(Toggle,1,SPARE_O510,SPARE_O510);
END_ROUTINE
